# EPICS substitutions: HeaterIoc/db/user.substitutions
# Example substitutions file

file "db/dbExample1.db" {
    { Heater = "hanlf",TMP_FB="hanlf:tempFeedbk",ALRM_TMP_FB="hanlf:alarmTempFB",PW_OUT="hanlf:powerOut" ,CTRL_OUT="hanlf:controlOut"}
}

file "db/dbExample2.db" {
    { Heater = "hanlf",TMP_FB="hanlf:tempFeedbk",ALRM_TMP_FB="hanlf:alarmTempFB",PW_OUT="hanlf:powerOut",CTRL_OUT="hanlf:controlOut" }
}
